{attribute 'qualified_only'}
VAR_GLOBAL
	TimeStartLigne  	: TIME;
	TimeStartMatch 		: TIME;
	TimeMatch 			: TIME;
	PointMatch 			: LREAL;
	MatchEnCours		: BOOL;

	Tableau 			: ARRAY[0..100] OF ST_Tableau;
	iLigne 				: INT;
	NextLigne			: BOOL;
	iCounter			: INT;
	
	bExecuteDeplacement : BOOL;
	bDeplacementFini	: BOOL;
	bActionFinie		: BOOL;
	
	iEtapeAction 		: INT := 0;
	iAsyncAction 		: STRING; 
END_VAR

(* stored: Version 1.1.0.1, ProductVersion 3.1.4024.12
   GVL G_Match: Id {60a8e4ef-30c4-40fc-80cf-b7b07ceed9bb} *)
